TYPE stSettings_AMR EXTENDS stSettings_Rob :
STRUCT
END_STRUCT
END_TYPE

(* stored: Version 1.1.0.1, ProductVersion 3.1.4026.18
   DUT stSettings_AMR: Id {c511243c-3394-41bc-9629-9ccadd27ffaf} *)
